FUNCTION_BLOCK FB_EstacionPreparar_SFC
VAR_INPUT
	//nuestras_variables
	Tcinta: TIME := T#0.5S;	

    // SFC-Flags
    SFCPause: BOOL;
    SFCReset: BOOL;

    // Indicadores de sincronizacion
    Ack: BOOL := TRUE;
    Execute: BOOL;

   //Entradas
    Horizontal_descargador_detras: BOOL;
	Vertical_descargador_arriba: BOOL;
	Presencia_pale: BOOL;
	
END_VAR
VAR_OUTPUT
    // Indicadores de sincronizacion
    Done: BOOL;
    Ready: BOOL;
	
	//Salidas
	Descargador_atras: BOOL;
	Activa_marcha_motor_cinta: BOOL;
END_VAR
VAR
END_VAR

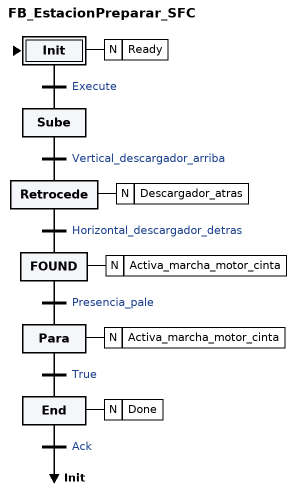
INITIAL_STEP Init:
    Ready(N);
END_STEP
TRANSITION FROM Init TO Sube
    := Execute;
END_TRANSITION
STEP Sube:
END_STEP
TRANSITION FROM Sube TO Retrocede
    := Vertical_descargador_arriba;
END_TRANSITION
STEP Retrocede:
    Descargador_atras(N);
END_STEP
TRANSITION FROM Retrocede TO FOUND
    := Horizontal_descargador_detras;
END_TRANSITION
STEP FOUND:
    Activa_marcha_motor_cinta(N);
END_STEP
TRANSITION FROM FOUND TO Para
    := Presencia_pale;
END_TRANSITION
STEP Para:
    Activa_marcha_motor_cinta(N);
END_STEP
TRANSITION FROM Para TO End
    := True;
END_TRANSITION
STEP End:
    Done(N);
END_STEP
TRANSITION FROM End TO Init
    := Ack;
END_TRANSITION

END_FUNCTION_BLOCK

(* stored: Version 1.1.0.1, ProductVersion 3.1.4024.12
   POU FB_EstacionPreparar_SFC: Id {b9eefe85-04a0-4d68-be74-7a048e2344ce}, SpecialFunc None *)
